{attribute 'hide_all_locals'}
FUNCTION_BLOCK FB_3_ROB_AXIS_LIN EXTENDS FB_2_ROB_AXIS

VAR
  _pSettingsLinAxis : POINTER TO stSettings_LinAxis;
END_VAR

CYCLIC_LIN_AXIS();

ACTION CYCLIC_LIN_AXIS:
IF _pSettingsLinAxis <> 0 THEN
  TCPPos_PLCUnit := _pSettingsLinAxis^.InstallationPose;
  TCPVel_PLCUnit.x := 0.0;
  TCPVel_PLCUnit.y := 0.0;
  TCPVel_PLCUnit.z := 0.0;

  CASE _pSettingsLinAxis^.Direction OF
    eDirections.Xplus:
      TCPPos_PLCUnit.x := TCPPos_PLCUnit.x + (ActualAxisPosition - _pSettingsLinAxis^.ZeroPosition);
      TCPVel_PLCUnit.x := _axisActualVelocity;
    eDirections.Xminus:
      TCPPos_PLCUnit.x := TCPPos_PLCUnit.x - (ActualAxisPosition - _pSettingsLinAxis^.ZeroPosition);
      TCPVel_PLCUnit.x := -_axisActualVelocity;
    eDirections.Yplus:
      TCPPos_PLCUnit.y := TCPPos_PLCUnit.y + (ActualAxisPosition - _pSettingsLinAxis^.ZeroPosition);
      TCPVel_PLCUnit.y := _axisActualVelocity;
    eDirections.Yminus:
      TCPPos_PLCUnit.y := TCPPos_PLCUnit.y - (ActualAxisPosition - _pSettingsLinAxis^.ZeroPosition);
      TCPVel_PLCUnit.y := -_axisActualVelocity;
    eDirections.Zplus:
      TCPPos_PLCUnit.z := TCPPos_PLCUnit.z + (ActualAxisPosition - _pSettingsLinAxis^.ZeroPosition);
      TCPVel_PLCUnit.z := _axisActualVelocity;
    eDirections.Zminus:
      TCPPos_PLCUnit.z := TCPPos_PLCUnit.z - (ActualAxisPosition - _pSettingsLinAxis^.ZeroPosition);
      TCPVel_PLCUnit.z := -_axisActualVelocity;
  END_CASE
END_IF

CYCLIC_AXIS();
END_ACTION

END_FUNCTION_BLOCK

(* stored: Version 1.1.0.1, ProductVersion 3.1.4026.18
   POU FB_3_ROB_AXIS_LIN: Id {0e318480-45bd-4a60-bef7-a58dd5c55756}, SpecialFunc None
   Action CYCLIC_LIN_AXIS: Id {5e1e5d5c-d399-452a-a592-785fd32ef430} *)
